FUNCTION_BLOCK Q_FontAttributes (* Command change font attributes ( Part 6 - F.28 ) *)
  (* Standard: ISO 11783-6; Description: Copyright (c) 2022 HR Agrartechnik GmbH This program and the accompanying materials are made available under the terms of the Eclipse Public License 2.0 which is available at https://www.eclipse.org/legal/epl-2.0/ SPDX-License-Identifier: EPL-2.0 see Description Tab *)
  (* Version 1.0, 2022-07-08, Franz Höpfinger, HR Agrartechnik GmbH *)
  PACKAGE isobus::UT::Q;
  IMPORT isobus::UT::Q::const::IDs::ID_NULL;
  (* Documentation:
  Command change font attributes ( Part 6 - F.28 )
   This command is used to change the font attributes in a font attributes object.
   Valid values for u16ObjId (the font attributes object)
   A font attributes Object ID is valid if it falls within the following ISO 11783-6 ID range (Annex F.28):
    - FontAttributesObject: 23000 – 23999
    ID_NULL (65535) is not a command target but can be used in INIT to deactivate the FB. Any ID outside this range is invalid for commanding.
   Activate / Deactivate
   The FB is deactivated by default. It becomes active when INIT provides a valid font attributes Object ID. Sending INIT with ID_NULL (65535) deactivates the FB again. This toggle can be repeated arbitrarily.
    - INIT + ID_NULL (65535): FB deactivated, STATUS="DEACTIVATED", s16result=VT_E_DEACTIVATED (-40)
   - INIT + valid font attributes ID: FB activated, STATUS="initialized", s16result=VT_E_NO_ERR (0). If a REQ was buffered before, it is executed immediately.
   - INIT + invalid ID: STATUS="ERROR: Invalid Object ID (not a font attributes object)", s16result=VT_E_INVALID_OBJECT_ID (-132)
    REQ Handling
    - REQ before any INIT: Buffered, STATUS="Buffered: INIT not yet completed", s16result=VT_E_NOT_READY (-131)
   - REQ while deactivated (INIT came with NULL or invalid ID): STATUS shows the actual deactivation reason, s16result=VT_E_DEACTIVATED (-40) or VT_E_INVALID_OBJECT_ID (-132)
   - REQ while active: Command sent to VT, result reflected in CNF
    param[in] {objectID, uint16_t}
   Object ID. Use ID_NULL (65535) to deactivate the FB. Use a valid font attributes object ID to activate.
   param[in] {colour, uint8_t}
   New font colour (see Part 6 - A.3)
   param[in] {size, uint8_t}
   New font size (see Part 6 - B.14)
   param[in] {type, uint8_t}
   New font type (see Part 6 - B.14)
   param[in] {styleBitfield, uint8_t}
   New font style (see Part 6 - B.14)
   Return Values (s16result):
   int16_t
    - VT_E_NO_ERR (0) - OK
   - VT_E_DEACTIVATED (-40) - FB deactivated (INIT received with ID_NULL)
   - VT_E_INVALID_OBJECT_ID (-132) - Object ID is invalid (not a font attributes object)
   - VT_E_NOT_READY (-131) - Buffered: INIT not yet completed
   - VT_E_OVERFLOW (-6) - buffer overflow
   - VT_E_NOACT (-8) - Command not possible in current state
   - VT_E_NO_INSTANCE (-21) - No VT client available
   - VT_E_ISO_INSTANCE_INVALID (-129) - Identifier for instance (connection) invalid
   - VT_E_NOT_ALIVE (-130) - Identifier for instance valid, but VT Dead.
    Instanz-Eindeutigkeit (Instance Uniqueness)
   Dieser Baustein erfordert Instanz-Eindeutigkeit bezüglich u16ObjId. Es darf im gesamten Programm nur eine Instanz von Q_FontAttributes für dieselbe Ziel-Objekt-ID existieren. Eine zweite Instanz auf dieselbe Objekt-ID wird bei INIT deaktiviert (STATUS = "This objID is already in use").
  *)
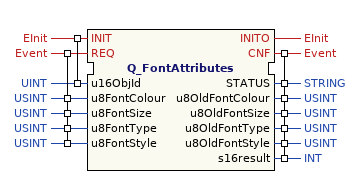
  EVENT_INPUT
    INIT : EInit WITH u16ObjId; (* Service Initialization *)
    REQ WITH u8FontColour, u8FontSize, u8FontType, u8FontStyle; (* Service Request *)
  END_EVENT
  EVENT_OUTPUT
    INITO : EInit; (* Initialization Confirm *)
    CNF WITH STATUS, u8OldFontType, u8OldFontColour, u8OldFontSize, s16result, u8OldFontStyle; (* Confirmation of Requested Service *)
  END_EVENT
  VAR_INPUT
    u16ObjId : UINT := ID_NULL; (* Object ID *)
    u8FontColour : USINT; (* New font colour (see Part 6 - A.3) *)
    u8FontSize : USINT; (* New font size (see Part 6 - B.14) *)
    u8FontType : USINT; (* New font type (see Part 6 - B.14) *)
    u8FontStyle : USINT; (* New font style (see Part 6 - B.14) *)
  END_VAR
  VAR_OUTPUT
    STATUS : STRING; (* Service Status *)
    u8OldFontColour : USINT; (* Old font colour (see Part 6 - A.3) *)
    u8OldFontSize : USINT; (* Old font size (see Part 6 - B.14) *)
    u8OldFontType : USINT; (* Old font type (see Part 6 - B.14) *)
    u8OldFontStyle : USINT; (* Old font style (see Part 6 - B.14) *)
    s16result : INT; (* retval see description *)
  END_VAR
END_FUNCTION_BLOCK
